FUNCTION Set_Buffer_Layout : Buffer_Error
VAR_INPUT
	Buffer_Size : USINT;
	Bool_Amount : USINT;
	Int_Amount : USINT;
	Real_Amount : USINT;
	String_Amount : USINT;
END_VAR

VAR_IN_OUT
	Layout : Buffer_Layout;
END_VAR

VAR
	ClearLayout : Buffer_Layout;
	CurrentSize : USINT := 0;
END_VAR

Layout.Buffer_Size := Buffer_Size;

IF Bool_Amount > 0 THEN
	ClearLayout.Bool_Amount := Bool_Amount;
	ClearLayout.Bool_Array_Offset := CurrentSize;
	ClearLayout.Enabel_Bool_Array := TRUE;
	CurrentSize := CurrentSize + (Bool_Amount * 1);
ELSE
	Layout.Enabel_Bool_Array := FALSE;
END_IF

IF Int_Amount > 0 THEN
	ClearLayout.Int_Amount := Int_Amount;
	ClearLayout.Int_Array_Offset := CurrentSize;
	ClearLayout.Enabel_Int_Array := TRUE;
	CurrentSize := CurrentSize + (Int_Amount * 2);
ELSE
	Layout.Enabel_Int_Array := FALSE;
END_IF

IF Real_Amount > 0 THEN
	ClearLayout.Real_Amount := Real_Amount;
	ClearLayout.Real_Array_Offset := CurrentSize;
	Layout.Enabel_Real_Array := TRUE;
	CurrentSize := CurrentSize + (Real_Amount * 4);
ELSE
	Layout.Enabel_Real_Array := FALSE;
END_IF

IF String_Amount > 0 THEN
	ClearLayout.String_Amount := String_Amount;
	ClearLayout.String_Array_Offset := CurrentSize;
	Layout.Enabel_String_Array := TRUE;
	CurrentSize := CurrentSize + (String_Amount * 8);
ELSE
	Layout.Enabel_String_Array := FALSE;
END_IF

IF Layout.Buffer_Size < Get_Layout_Size(Layout:= ClearLayout) THEN
	Set_Buffer_Layout := Buffer_Error.Overflow;
ELSE
	Layout := ClearLayout;
	Set_Buffer_Layout := Buffer_Error.None;
END_IF

END_FUNCTION

(* stored: Version 1.1.0.1, ProductVersion 3.1.4024.10
   POU Set_Buffer_Layout: Id {6f5bf570-96c4-4372-a41d-eb5b698ff879}, SpecialFunc None *)
